FUNCTION_BLOCK FB_estop EXTENDS FB_pushBtnNC
VAR
	bResetEstopFb 		AT %Q* : BOOL;
	bEstopFbError 		AT %I* : BOOL;
	bEstopSigOk 		AT %I* : BOOL;
	nEstopFbState		AT %I* : USINT; //States : 1 - Running, 2 - PreOp, 3 - Triggered, 6 - Reset 
END_VAR

METHOD reset : BOOL
VAR_INPUT
END_VAR
reset := FALSE;
bResetEstopFb := TRUE;
IF NOT bEstopFbError THEN
	bResetEstopFb := FALSE;
	reset := TRUE;
END_IF
END_METHOD

PROPERTY resetEstopFB : BOOL
SET
bResetEstopFb := resetEstopFB;
END_SET
END_PROPERTY

END_FUNCTION_BLOCK

(* stored: Version 1.1.0.1, ProductVersion 3.1.4024.13
   POU FB_estop: Id {17167641-fb84-44e0-a1b5-cde62190fc72}, SpecialFunc None
   Method reset: Id {a2f857f7-8c32-4efc-aee1-ece786c7f1b3}
   Property resetEstopFB: Id {e841fe5c-79b0-47db-aca0-2bbc1160c0a2}
   Set Set: Id {f359c5cd-0778-4107-8338-d864b4e712c5} *)
